// TwinCAT 3 PLC project CX2040_PLC
// ProgramVersion: 3.1.4023.0
// libraries:
//   Tc2_Standard, * (Beckhoff Automation GmbH)
//   Tc2_System, * (Beckhoff Automation GmbH)
//   Tc3_Module, * (Beckhoff Automation GmbH)
// project tree:
//   GVLs/ GVL.TcGVL
//   / PlcTask.TcTTO
//   POUs/ MAIN.TcPOU

CONFIGURATION CX2040_PLC
    RESOURCE PLC ON TwinCAT3
        TASK PlcTask(INTERVAL := T#1ms, PRIORITY := 20);
        PROGRAM MAIN WITH PlcTask : MAIN;
    END_RESOURCE
END_CONFIGURATION

// ---- GVLs/GVL.TcGVL
{attribute 'qualified_only'}
VAR_GLOBAL
	bIn AT %I* : BOOL;
	bOut AT %Q* : BOOL;
	
	iIn AT %I* : USINT;
	iOut AT %Q* : USINT;
END_VAR

// ---- POUs/MAIN.TcPOU
PROGRAM MAIN
VAR
	bIn : BOOL;
	bOut : BOOL;
END_VAR

bIn := GVL.bIn;

GVL.bOut := bOut;

END_PROGRAM
